(* Logix 5000 project; controller FRIST_EXAMPLE Emulate 5570 rev 19.11; software revision 19.01 *)

TASK MainTask (continuous, watchdog 500 ms) : MainProgram

MODULES
   Local : Emulate 5570 (ICP 2, rev 19.11)
       : 1756-IB32 (ICP 3, rev 3.1, Input RPI 20 ms)   // DG-INPUT
       : vendor 1 type 7 code 8 (ICP 4, rev 3.1, Output RPI 20 ms)
       : 1756-IF6I (ICP 5, rev 1.1, Input RPI 100 ms)
       : 1756-OF8 (ICP 6, rev 1.1, Output RPI 12 ms)
END_MODULES

VAR_GLOBAL   (* controller tags *)
   CMD_MT01 : BOOL;
   DESLIGA : BOOL := 1;
   LIGA : BOOL;
END_VAR

PROGRAM MainProgram   (* main routine MainRoutine *)
VAR
   FIT01 : REAL;
   PID_CONTROL : PID := (MAXS := 100.0, MAXO := 100.0, UPD := 0.1, MAXI := 100.0, MAXCV := 100.0, MAXTIE := 100.0);
   VAL01 : REAL;
END_VAR

ROUTINE MainRoutine   (* ladder *)
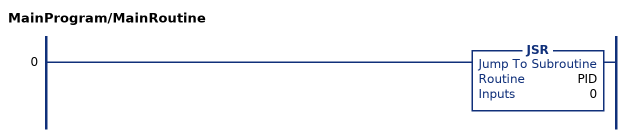
   0: JSR(PID,0);
END_ROUTINE

ROUTINE PID   (* ladder *)
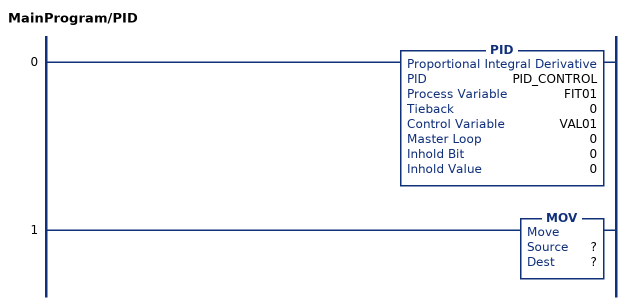
   0: PID(PID_CONTROL,FIT01,0,VAL01,0,0,0);
   1: MOV(?,?);
END_ROUTINE
END_PROGRAM
